METHOD PRIVATE CheckImplementsIList
VAR
	list : List;
    iList : I_List := list;
    result : BOOL;
END_VAR
TEST('ListTests_CheckImplementsIList');

result := iList <> 0;

AssertTrue(Condition := result,
    Message := 'Did not implement IList');

TEST_FINISHED();
END_METHOD

METHOD PUBLIC CheckIsEmptyWhenEmpty
VAR
	result : BOOL;
	list : List;
END_VAR
TEST('CheckIsEmptyWhenEmpty');

// @TEST-RUN
result := list.IsEmpty;

// @TEST-ASSSERT
AssertTrue(
	Condition := result,
	Message := 'Incorrect state of IsEmpty'
);

TEST_FINISHED();
END_METHOD

METHOD PUBLIC CheckIsEmptyWhenFull
VAR
	in : INT := 123;
	result : BOOL;
	list : List;
END_VAR
TEST('CheckIsEmptyWhenFull');

// @TEST-FIXTURE
list.AddItem(in);

// @TEST-RUN
result := list.IsEmpty;

// @TEST-ASSSERT
AssertFalse(
	Condition := result,
	Message := 'Incorrect state of IsEmpty'
);

TEST_FINISHED();
END_METHOD

METHOD PUBLIC CheckOffEvent
VAR
	value : INT := 123;
	list : List;
	handler : CollectionChangedEventHandler(ExpectedOriginator := list);
END_VAR
TEST('CheckOffEvent');

// @TEST-FIXTURE
list.OnEvent('OnChanged',handler);
list.OffEvent('OnChanged',handler);

// @TEST-RUN
list.AddItem(value);

// @TEST-ASSSERT
AssertFalse(
	Condition := handler.EventReceived,
	Message := 'OnceEvent emitted the OnChanged event more than once'
);

TEST_FINISHED();
END_METHOD

METHOD PUBLIC CheckOnceEvent
VAR
	value : INT := 123;
	list : List;
	handler : CollectionChangedEventHandler(ExpectedOriginator := list);
END_VAR
TEST('CheckOnceEvent');

// @TEST-FIXTURE
list.OnceEvent('OnChanged',handler);
list.AddItem(value);
handler.Reset();

// @TEST-RUN
list.AddItem(value);

// @TEST-ASSSERT
AssertFalse(
	Condition := handler.EventReceived,
	Message := 'OnceEvent emitted the OnChanged event more than once'
);

TEST_FINISHED();
END_METHOD

METHOD PUBLIC CheckOnChangedEvent
VAR
	value : INT := 123;
	list : List;
	handler : CollectionChangedEventHandler(ExpectedOriginator := list);
END_VAR
TEST('CheckOnChangedEvent');

// @TEST-FIXTURE
list.OnEvent('OnChanged',handler);

// @TEST-RUN
list.AddItem(value);

// @TEST-ASSSERT
AssertTrue(
	Condition := handler.EventReceived,
	Message := 'Did not emit the OnChanged event'
);

AssertTrue(
	Condition := handler.FromExpectedOriginator,
	Message := 'Did not include itself in the OnChanged event'
);

TEST_FINISHED();
END_METHOD

METHOD PUBLIC CheckOnDisposedEvent
VAR
	pList : POINTER TO List;
	handler : CollectionDisposedEventHandler(ExpectedOriginator := 0);
END_VAR
TEST('CheckOnDisposedEvent');

// @TEST-FIXTURE
pList := __NEW(List);
handler.SetExpectedOriginator(pList^);
pList^.OnEvent('OnDisposed',handler);

// @TEST-RUN
pList^.Dispose();

// @TEST-ASSSERT
AssertTrue(
	Condition := handler.EventReceived,
	Message := 'Did not emit the OnDisposed event'
);

AssertTrue(
	Condition := handler.FromExpectedOriginator,
	Message := 'Did not include itself in the OnDisposed event'
);

TEST_FINISHED();
END_METHOD

METHOD PRIVATE CheckTrimExcessAfterAdding5Items
VAR
	in1 : INT := 1;
	in2 : INT := 2;
	in3 : INT := 3;
	in4 : INT := 4;
	in5 : INT := 5;
	in6 : INT := 6;
	expected : DINT := 5;
	out : DINT;
	list : List;
END_VAR
TEST('CheckTrimExcessAfterAdding5Items');

list.AddItem(in1); // [1, null, null, null]
list.AddItem(in2); // [1, 2, null, null]
list.AddItem(in3); // [1, 2, 3, null]
list.AddItem(in4); // [1, 2, 3, 4]
list.AddItem(in5); // [1, 2, 3, 4, 5, null, null, null]
list.TrimExcess(); // [1, 2, 3, 4, 5]

out := list.Capacity;

AssertEquals(expected, out, 'List was expected to double once 5 items were added');

TEST_FINISHED();
END_METHOD

METHOD PRIVATE CheckTryCopyTo
VAR
	in1 : INT := 123;
	in2 : INT := 456;
	in3 : INT := 789;
	out : ARRAY [0..2] OF INT;
	expected : ARRAY [0..2] OF INT := [123,456,789];
	list : List;
END_VAR
TEST('CheckTryCopyTo');

list.AddItem(in1); // [123]
list.AddItem(in2); // [123,456]
list.AddItem(in3); // [123,456,789]

list.TryCopyTo(out);

AssertEquals(
	Expected := expected,
	Actual := out,
	Message := 'Did not produce the expected result'
);

TEST_FINISHED();
END_METHOD

METHOD PRIVATE CheckTryCopyToLocation
VAR
	in1 : INT := 123;
	in2 : INT := 456;
	in3 : INT := 789;
	out : ARRAY [0..2] OF INT;
	expected : ARRAY [0..2] OF INT := [123,456,789];
	list : List;
END_VAR
TEST('CheckTryCopyToLocation');

list.AddItem(in1); // [123]
list.AddItem(in2); // [123,456]
list.AddItem(in3); // [123,456,789]

list.TryCopyToLocation(ADR(out),SIZEOF(out));

AssertEquals(
	Expected := expected,
	Actual := out,
	Message := 'Did not produce the expected result'
);

TEST_FINISHED();
END_METHOD

METHOD PRIVATE CheckTryInsert
VAR
	in1 : INT := 123;
	in2 : INT := 456;
	in3 : INT := 789;
	out : INT;
	result : BOOL;
	expected : INT := 789;
	list : List;
END_VAR
TEST('CheckTryInsert');

list.AddItem(in1); // [123]
list.AddItem(in1); // [123,456]
list.TryInsert(1, in3); // [123,789,456]

list.TryGetByIndex(1,out);

AssertEquals(expected, out, 'Did not produce the expected result');

TEST_FINISHED();
END_METHOD

METHOD PRIVATE CheckTryRemoveAtInBounds
VAR
	in1 : INT := 123;
	in2 : INT := 456;
	in3 : INT := 789;
	out : INT;
	result : BOOL;
	list : List;
END_VAR
TEST('CheckTryRemoveAtInBounds');

list.AddItem(in1); // [123]
list.AddItem(in2); // [123,456]
list.AddItem(in3); // [123,456,789]

list.TryRemoveAt(0);

result := list.TryGetByIndex(0, out);

AssertTrue(result, 'Couldnt get first item');
AssertEquals(in2, out, 'Array didnt shift up items');

TEST_FINISHED();
END_METHOD

METHOD PRIVATE CheckTryRemoveAtNoItems
VAR
	out : INT;
	result : BOOL;
	list : List;
END_VAR
TEST('CheckTryRemoveAtNoItems');

result := list.TryRemoveAt(0);

AssertFalse(result, 'Returned true while there was nothing to remove');

TEST_FINISHED();
END_METHOD

METHOD PRIVATE CheckTryRemoveAtOutOfBounds
VAR
	in1 : INT := 123;
	in2 : INT := 456;
	in3 : INT := 789;
	out : INT;
	result : BOOL;
	list : List;
END_VAR
TEST('CheckTryRemoveAtOutOfBounds');

list.AddItem(in1); // [123]
list.AddItem(in2); // [123,456]
list.AddItem(in3); // [123,456,789]

result := list.TryRemoveAt(3);

AssertFalse(result, 'Returned true while remove was out of bounds');

TEST_FINISHED();
END_METHOD

METHOD PRIVATE CheckTryRemoveItemFirstShiftUp
VAR
	in1 : INT := 123;
	in2 : INT := 456;
	in3 : INT := 789;
	out : INT;
	result : BOOL;
	expected : INT := 456;
	list : List;
END_VAR
TEST('CheckTryRemoveItemFirstShiftUp');

list.AddItem(in1); // [123]
list.AddItem(in2); // [123,456]
list.AddItem(in3); // [123,456,789]
list.TryRemoveItem(in1); // [456,789]

result := list.TryGetByIndex(0, out);

AssertTrue(result, 'Couldnt get first item');

AssertEquals(expected, out, 'Array didnt shift up items');

TEST_FINISHED();
END_METHOD

METHOD PRIVATE CheckTryRemoveItemNonExisting
VAR
	in1 : INT := 123;
	in2 : INT := 456;
	in3 : INT := 789;
	out : INT;
	result : BOOL;
	list : List;
END_VAR
TEST('CheckTryRemoveItemNonExisting');

list.AddItem(in1); // [123]
list.AddItem(in2); // [123,456]

result := list.TryRemoveItem(in3);

AssertFalse(result, 'RemoveItem returned true which should not happen when item does not exist');

TEST_FINISHED();
END_METHOD

METHOD PRIVATE CheckTryRemoveItemSecondShiftUp
VAR
	in1 : INT := 123;
	in2 : INT := 456;
	in3 : INT := 789;
	out : INT;
	result : BOOL;
	expected : INT := 789;
	list : List;
END_VAR
TEST('CheckTryRemoveItemSecondShiftUp');

list.AddItem(in1); // [123]
list.AddItem(in2); // [123,456]
list.AddItem(in3); // [123,456,789]
list.TryRemoveItem(in2); // [123,789]

result := list.TryGetByIndex(1, out);

AssertTrue(result, 'Coulndt get first item');
AssertEquals(expected, out, 'Array didnt shift up items');

TEST_FINISHED();
END_METHOD

END_FUNCTION_BLOCK

// ---- Tests/ListForwardEnumerator_TestSuite.TcPOU
FUNCTION_BLOCK ListForwardEnumerator_TestSuite EXTENDS TcUnit.FB_TestSuite
VAR
END_VAR

CheckIsValidAtStart();
CheckMoveNextReturnsFalseAtTheEnd();
CheckMoveNextReturnsTrueSingleItem();
CheckMoveNextReturnsFalseWhenEmpty();
CheckMoveNextReturnsTrueMultipleItems();
CheckReset();
CheckTryGet();
CheckTryGetTo();
CheckWorksWithArrays();
CheckWorksWithIntegers();
CheckWorksWithStrings();

METHOD PRIVATE CheckIsValidAtStart
VAR
	result : BOOL;
	store : List;
	enumerator : I_ForwardEnumerator;
END_VAR
TEST('CheckIsValidAtStart');

enumerator := store.GetEnumerator();

result := enumerator.IsValid;
enumerator.Dispose();

AssertTrue(
	Condition := result,
	Message := 'IsValid returned false'
);

TEST_FINISHED();
END_METHOD

METHOD PRIVATE CheckMoveNextReturnsFalseAtTheEnd
VAR
	in1 : INT := 123;
	result : BOOL;
	store : List;
	enumerator : I_ForwardEnumerator;
END_VAR
TEST('CheckMoveNextReturnsFalseAtTheEnd');

store.AddItem(in1);
enumerator := store.GetEnumerator();

enumerator.MoveNext();
result := enumerator.MoveNext();
enumerator.Dispose();

AssertFalse(result,
    'MoveNext did not correctly signal the end of the enumeration');
	
TEST_FINISHED();
END_METHOD

METHOD PRIVATE CheckMoveNextReturnsFalseWhenEmpty
VAR
	result : BOOL;
	store : List;
	enumerator : I_ForwardEnumerator;
	count : DINT;
END_VAR
TEST('CheckMoveNextReturnsFalseWhenEmpty');

count := store.Count;
enumerator := store.GetEnumerator();

result := enumerator.MoveNext();
enumerator.Dispose();

AssertFalse(Condition := result,
    Message := 'MoveNext did not correctly signal the end of the enumeration');

TEST_FINISHED();
END_METHOD

METHOD PRIVATE CheckMoveNextReturnsTrueMultipleItems
VAR
	in1 : INT := 123;
	in2 : INT := 456;
	in3 : INT := 789;
	result : BOOL;
	store : List;
	enumerator : I_ForwardEnumerator;
END_VAR
TEST('CheckMoveNextReturnsTrueMultipleItems');

store.AddItem(in1);
store.AddItem(in2);
store.AddItem(in3);
enumerator := store.GetEnumerator();

result := enumerator.MoveNext();
enumerator.Dispose();

AssertTrue(result, 'MoveNext did not correctly signal there were more items to follow');

TEST_FINISHED();
END_METHOD

METHOD PRIVATE CheckMoveNextReturnsTrueSingleItem
VAR
	in1 : INT := 123;
	result : BOOL;
	store : List;
	enumerator : I_ForwardEnumerator;
END_VAR
TEST('CheckMoveNextReturnsTrueSingleItem');

store.AddItem(in1);
enumerator := store.GetEnumerator();

result := enumerator.MoveNext();
enumerator.Dispose();

AssertTrue(result,
    'MoveNext did not correctly signal there were more items to follow');
	
TEST_FINISHED();
END_METHOD

METHOD PRIVATE CheckReset
VAR
	in1 : ARRAY [0..1] OF REAL := [0.1,2.3];
	in2 : ARRAY [0..1] OF REAL := [1.2,3.4];
	in3 : ARRAY [0..1] OF REAL := [2.3,4.5];
	out : ARRAY [0..1] OF REAL;
	expected : ARRAY [0..1] OF REAL := [0.1,2.3];
	store : List;
	enumerator : I_ForwardEnumerator;
END_VAR
TEST('CheckReset');

store.AddItem(in1);
store.AddItem(in2);
store.AddItem(in3);

enumerator := store.GetEnumerator();

enumerator.MoveNext();
enumerator.MoveNext();
enumerator.Reset();
enumerator.MoveNext();
enumerator.TryGet(out);

enumerator.Dispose();

AssertEquals(
	Expected := expected,
	Actual := out,
	Message := 'Did not produce the expected result'
);

TEST_FINISHED();
END_METHOD

METHOD PRIVATE CheckTryGet
VAR
	in : INT := 123;
	out : INT;
	expected : INT := 123;
	result : BOOL;
	store : List;
	enumerator : I_ForwardEnumerator;
END_VAR
TEST('CheckTryGet');

store.AddItem(in);
enumerator := store.GetEnumerator();
enumerator.MoveNext();

result := enumerator.TryGet(out);
enumerator.Dispose();

AssertTrue(
	Condition := result,
	Message := 'Method returned false'
);

AssertEquals(
	Expected := expected,
	Actual := out,
	Message := 'Did not produce the expected result'
);

TEST_FINISHED();
END_METHOD

METHOD PRIVATE CheckTryGetTo
VAR
	in : INT := 123;
	out : INT;
	expected : INT := 123;
	result : BOOL;
	store : List;
	enumerator : I_ForwardEnumerator;
END_VAR
TEST('CheckTryGetTo');

store.AddItem(in);
enumerator := store.GetEnumerator();
enumerator.MoveNext();

result := enumerator.TryGetTo(ADR(out),SIZEOF(out));
enumerator.Dispose();

AssertTrue(
	Condition := result,
	Message := 'Method returned false'
);

AssertEquals(
	Expected := expected,
	Actual := out,
	Message := 'Did not produce the expected result'
);

TEST_FINISHED();
END_METHOD

METHOD PRIVATE CheckWorksWithArrays
VAR
	in1 : ARRAY [0..1] OF REAL := [0.1,2.3];
	in2 : ARRAY [0..1] OF REAL := [1.2,3.4];
	in3 : ARRAY [0..1] OF REAL := [2.3,4.5];
	out1 : ARRAY [0..1] OF REAL;
	out2 : ARRAY [0..1] OF REAL;
	out3 : ARRAY [0..1] OF REAL;
	expected1 : ARRAY [0..1] OF REAL := [0.1,2.3];
	expected2 : ARRAY [0..1] OF REAL := [1.2,3.4];
	expected3 : ARRAY [0..1] OF REAL := [2.3,4.5];
	store : List;
	enumerator : I_ForwardEnumerator;
END_VAR
TEST('CheckWorksWithArrays');

store.AddItem(in1);
store.AddItem(in2);
store.AddItem(in3);

enumerator := store.GetEnumerator();

enumerator.MoveNext();
enumerator.TryGet(out1);
enumerator.MoveNext();
enumerator.TryGet(out2);
enumerator.MoveNext();
enumerator.TryGet(out3);

enumerator.Dispose();

AssertEquals(
	Expected := expected1,
	Actual := out1,
	Message := 'Did not produce the expected 1st result'
);

AssertEquals(
	Expected := expected2,
	Actual := out2,
	Message := 'Did not produce the expected 2nd result'
);

AssertEquals(
	Expected := expected3,
	Actual := out3,
	Message := 'Did not produce the expected 3rd result'
);

TEST_FINISHED();
END_METHOD

METHOD PRIVATE CheckWorksWithIntegers
VAR
	in1 : INT := 123;
	in2 : INT := 234;
	in3 : INT := 345;
	out1 : INT;
	out2 : INT;
	out3 : INT;
	expected1 : INT := 123;
	expected2 : INT := 234;
	expected3 : INT := 345;
	store : List;
	enumerator : I_ForwardEnumerator;
END_VAR
TEST('CheckWorksWithIntegers');

store.AddItem(in1);
store.AddItem(in2);
store.AddItem(in3);

enumerator := store.GetEnumerator();

enumerator.MoveNext();
enumerator.TryGet(out1);
enumerator.MoveNext();
enumerator.TryGet(out2);
enumerator.MoveNext();
enumerator.TryGet(out3);

enumerator.Dispose();

AssertEquals(
	Expected := expected1,
	Actual := out1,
	Message := 'Did not produce the expected 1st result'
);

AssertEquals(
	Expected := expected2,
	Actual := out2,
	Message := 'Did not produce the expected 2nd result'
);

AssertEquals(
	Expected := expected3,
	Actual := out3,
	Message := 'Did not produce the expected 3rd result'
);

TEST_FINISHED();
END_METHOD

METHOD PRIVATE CheckWorksWithStrings
VAR
	in1 : STRING := 'test1';
	in2 : STRING := 'test2';
	in3 : STRING := 'test3';
	out1 : STRING;
	out2 : STRING;
	out3 : STRING;
	expected1 : STRING := 'test1';
	expected2 : STRING := 'test2';
	expected3 : STRING := 'test3';
	store : List;
	enumerator : I_ForwardEnumerator;
END_VAR
TEST('CheckWorksWithStrings');

store.AddItem(in1);
store.AddItem(in2);
store.AddItem(in3);

enumerator := store.GetEnumerator();

enumerator.MoveNext();
enumerator.TryGet(out1);
enumerator.MoveNext();
enumerator.TryGet(out2);
enumerator.MoveNext();
enumerator.TryGet(out3);

enumerator.Dispose();

AssertEquals(
	Expected := expected1,
	Actual := out1,
	Message := 'Did not produce the expected 1st result'
);

AssertEquals(
	Expected := expected2,
	Actual := out2,
	Message := 'Did not produce the expected 2nd result'
);

AssertEquals(
	Expected := expected3,
	Actual := out3,
	Message := 'Did not produce the expected 3rd result'
);

TEST_FINISHED();
END_METHOD

END_FUNCTION_BLOCK

// ---- Tests/Queue_TestSuite.TcPOU
FUNCTION_BLOCK PUBLIC Queue_TestSuite EXTENDS TcUnit.FB_TestSuite

// check datatypes are handled correctly
CheckListWorksWithIntegers();
CheckListWorksWithStrings();
CheckListWorksWithArrays();

// all other checks
CheckQueueImplementsI_Queue();
CheckContains();
CheckClear();
CheckCount();
CheckAddItem();
CheckTryRemoveItem();
CheckTryDequeueRemovesTheItem();
CheckTryDequeueReturnsTheCorrectValue();
CheckTryPeekReturnsTheCorrectValue();
CheckTryPeekDoesNotRemoveTheItem();
CheckOnChangedEvent();
CheckOnDisposedEvent();
CheckOnceEvent();
CheckOffEvent();
CheckTryCopyTo();
CheckTryCopyToLocation();
CheckQueueOrderIsCorrect();
CheckListReturnsEnumerator();
CheckEnumeratorIsInvalidAfterChange();
CheckIsEmptyWhenEmpty();
CheckIsEmptyWhenFull();

METHOD PUBLIC CheckAddItem
VAR
	in1 : INT := 123;
	in2 : INT := 456;
	in3 : INT := 789;
	result : BOOL;
	queue : Queue;
END_VAR
TEST('CheckAddItem');

// @TEST-FIXTURE
queue.Enqueue(in1); // (lifo->) 123
queue.Enqueue(in2); // (lifo->) 123, 456

// @TEST-RUN
queue.AddItem(in3); // (lifo->) 123, 456, 789
result := queue.Contains(in3);

// @TEST-ASSSERT
AssertTrue(
	Condition := result,
	Message := 'Method returned false'
);

TEST_FINISHED();
END_METHOD

METHOD PUBLIC CheckClear
VAR
	in1 : INT := 123;
	in2 : INT := 456;
	in3 : INT := 789;
	queue : Queue;
END_VAR
TEST('CheckClear');

// @TEST-FIXTURE
queue.Enqueue(in1); // (lifo->) 123
queue.Enqueue(in2); // (lifo->) 123, 456
queue.Enqueue(in2); // (lifo->) 123, 456, 789

// @TEST-RUN
queue.Clear();

// @TEST-ASSSERT
AssertTrue(
	Condition := queue.Count = 0,
	Message := 'The count is not zero'
);

TEST_FINISHED();
END_METHOD

METHOD PUBLIC CheckContains
VAR
	in1 : INT := 123;
	in2 : INT := 456;
	in3 : INT := 789;
	result : BOOL;
	queue : Queue;
END_VAR
TEST('CheckContains');

// @TEST-FIXTURE
queue.Enqueue(in1); // (lifo->) 123
queue.Enqueue(in2); // (lifo->) 123, 456
queue.Enqueue(in2); // (lifo->) 123, 456, 789

// @TEST-RUN
result := queue.Contains(in2);

// @TEST-ASSSERT
AssertTrue(
	Condition := result,
	Message := 'Did not find the item in the queue'
);

TEST_FINISHED();
END_METHOD

METHOD PUBLIC CheckCount
VAR
	in1 : INT := 123;
	in2 : INT := 456;
	in3 : INT := 789;
	total : DINT;
	expected : DINT := 3;
	queue : Queue;
END_VAR
TEST('CheckCount');

// @TEST-FIXTURE
queue.Enqueue(in1); // (lifo->) 123
queue.Enqueue(in2); // (lifo->) 123, 456
queue.Enqueue(in2); // (lifo->) 123, 456, 789

// @TEST-RUN
total := queue.Count;

// @TEST-ASSSERT
AssertEquals(
	Expected := expected,
	Actual := total,
	Message := 'Incorrect count'
);

TEST_FINISHED();
END_METHOD

METHOD PUBLIC CheckEnumeratorIsInvalidAfterChange
VAR
	in : INT := 123;
	result : BOOL;
	queue : Queue;
	enumerator : I_ForwardEnumerator;
END_VAR
TEST('CheckEnumeratorIsInvalidAfterChange');

// @TEST-FIXTURE
enumerator := queue.GetEnumerator();
queue.Enqueue(in);

// @TEST-RUN
result := enumerator.IsValid;
enumerator.Dispose();

// @TEST-ASSSERT
AssertFalse(
	Condition := result,
	Message := 'Method returned true'
);

TEST_FINISHED();
END_METHOD

METHOD PUBLIC CheckIsEmptyWhenEmpty
VAR
	result : BOOL;
	queue : Queue;
END_VAR
TEST('CheckIsEmptyWhenEmpty');

// @TEST-RUN
result := queue.IsEmpty;

// @TEST-ASSSERT
AssertTrue(
	Condition := result,
	Message := 'Incorrect state of IsEmpty'
);

TEST_FINISHED();
END_METHOD

METHOD PUBLIC CheckIsEmptyWhenFull
VAR
	in : INT := 123;
	result : BOOL;
	queue : Queue;
END_VAR
TEST('CheckIsEmptyWhenFull');

// @TEST-FIXTURE
queue.Enqueue(in);

// @TEST-RUN
result := queue.IsEmpty;

// @TEST-ASSSERT
AssertFalse(
	Condition := result,
	Message := 'Incorrect state of IsEmpty'
);

TEST_FINISHED();
END_METHOD

METHOD PUBLIC CheckListReturnsEnumerator
VAR
	in1 : INT := 123;
	in2 : INT := 456;
	in3 : INT := 789;
	enumerator : I_ForwardEnumerator;
	queue : Queue;
END_VAR
TEST('CheckListReturnsEnumerator');

// @TEST-FIXTURE
queue.Enqueue(in1); // (lifo->) 123
queue.Enqueue(in2); // (lifo->) 123, 456
queue.Enqueue(in2); // (lifo->) 123, 456, 789

// @TEST-RUN
enumerator := queue.GetEnumerator();

// @TEST-ASSSERT
AssertTrue(
	Condition := (enumerator <> 0),
	Message := 'Did not return an enumerator'
);

// @TEST-DISPOSE
enumerator.Dispose();

TEST_FINISHED();
END_METHOD

METHOD PUBLIC CheckListWorksWithArrays
VAR
	in : ARRAY [0..1] OF REAL := [0.1,2.3];
	out : ARRAY [0..1] OF REAL;
	expected : ARRAY [0..1] OF REAL := [0.1,2.3];
	result : BOOL;
	queue : Queue;
END_VAR
TEST('CheckListWorksWithArrays');

// @TEST-FIXTURE
queue.Enqueue(in);

// @TEST-RUN
result := queue.TryDequeue(out);

// @TEST-ASSSERT
AssertTrue(
	Condition := result,
	Message := 'Method returned false'
);

AssertEquals(
	Expected := expected,
	Actual := out,
	Message := 'Did not produce the expected result'
);

TEST_FINISHED();
END_METHOD

METHOD PUBLIC CheckListWorksWithIntegers
VAR
	in : INT := 123;
	out : INT;
	expected : INT := 123;
	result : BOOL;
	queue : Queue;
END_VAR
TEST('CheckListWorksWithIntegers');

// @TEST-FIXTURE
queue.Enqueue(in);

// @TEST-RUN
result := queue.TryDequeue(out);

// @TEST-ASSSERT
AssertTrue(
	Condition := result,
	Message := 'Method returned false'
);

AssertEquals(
	Expected := expected,
	Actual := out,
	Message := 'Did not produce the expected result'
);

TEST_FINISHED();
END_METHOD

METHOD PUBLIC CheckListWorksWithStrings
VAR
	in : STRING := 'test';
	out : STRING;
	expected : STRING := 'test';
	result : BOOL;
	queue : Queue;
END_VAR
TEST('CheckListWorksWithStrings');

// @TEST-FIXTURE
queue.Enqueue(in);

// @TEST-RUN
result := queue.TryDequeue(out);

// @TEST-ASSSERT
AssertTrue(
	Condition := result,
	Message := 'Method returned false'
);

AssertEquals(
	Expected := expected,
	Actual := out,
	Message := 'Did not produce the expected result'
);

TEST_FINISHED();
END_METHOD

METHOD PUBLIC CheckOffEvent
VAR
	value : INT := 123;
	queue : queue;
	handler : CollectionChangedEventHandler(ExpectedOriginator := queue);
END_VAR
TEST('CheckOffEvent');

// @TEST-FIXTURE
queue.OnEvent('OnChanged',handler);
queue.OffEvent('OnChanged',handler);

// @TEST-RUN
queue.Enqueue(value);

// @TEST-ASSSERT
AssertFalse(
	Condition := handler.EventReceived,
	Message := 'OnceEvent emitted the OnChanged event more than once'
);

TEST_FINISHED();
END_METHOD

METHOD PUBLIC CheckOnceEvent
VAR
	value : INT := 123;
	queue : Queue;
	handler : CollectionChangedEventHandler(ExpectedOriginator := queue);
END_VAR
TEST('CheckOnceEvent');

// @TEST-FIXTURE
queue.OnceEvent('OnChanged',handler);
queue.Enqueue(value);
handler.Reset();

// @TEST-RUN
queue.Enqueue(value);

// @TEST-ASSSERT
AssertFalse(
	Condition := handler.EventReceived,
	Message := 'OnceEvent emitted the OnChanged event more than once'
);

TEST_FINISHED();
END_METHOD

METHOD PUBLIC CheckOnChangedEvent
VAR
	value : INT := 123;
	queue : Queue;
	handler : CollectionChangedEventHandler(ExpectedOriginator := queue);
END_VAR
TEST('CheckOnChangedEvent');

// @TEST-FIXTURE
queue.OnEvent('OnChanged', handler);

// @TEST-RUN
queue.Enqueue(value);

// @TEST-ASSSERT
AssertTrue(
	Condition := handler.EventReceived,
	Message := 'Did not emit the OnChanged event'
);

AssertTrue(
	Condition := handler.FromExpectedOriginator,
	Message := 'Did not include itself in the OnChanged event'
);

TEST_FINISHED();
END_METHOD

METHOD PUBLIC CheckOnDisposedEvent
VAR
	value : INT := 123;
	pQueue : POINTER TO Queue;
	handler : CollectionDisposedEventHandler(ExpectedOriginator := 0);
END_VAR
TEST('CheckOnDisposedEvent');

// @TEST-FIXTURE
pQueue := __NEW(Queue);
handler.SetExpectedOriginator(pQueue^);
pQueue^.OnEvent('OnDisposed', handler);

// @TEST-RUN
pQueue^.Dispose();

// @TEST-ASSSERT
AssertTrue(
	Condition := handler.EventReceived,
	Message := 'Did not emit the OnDisposed event'
);

AssertTrue(
	Condition := handler.FromExpectedOriginator,
	Message := 'Did not include itself in the OnDisposed event'
);

TEST_FINISHED();
END_METHOD

METHOD PUBLIC CheckQueueImplementsI_Queue
VAR
	queue : Queue;
    iQueue : I_Queue := queue;
    result : BOOL;
END_VAR
TEST('CheckQueueImplementsI_Queue');

// @TEST-FIXTURE

// @TEST-RUN
result := iQueue <> 0;

// @TEST-ASSSERT
AssertTrue(
	Condition := result,
	Message := 'Did not implement I_Queue'
);

TEST_FINISHED();
END_METHOD

METHOD PUBLIC CheckQueueOrderIsCorrect
VAR
	in1 : INT := 123;
	in2 : INT := 456;
	in3 : INT := 789;
	out1, out2, out3 : INT;
	expected1 : INT := 123;
	expected2 : INT := 456;
	expected3 : INT := 789;
	result1, result2, result3 : BOOL;
	queue : Queue;
END_VAR
TEST('CheckQueueOrderIsCorrect');

// @TEST-FIXTURE
queue.Enqueue(in1); // (lifo->) 123
queue.Enqueue(in2); // (lifo->) 123, 456
queue.Enqueue(in3); // (lifo->) 123, 456, 789

// @TEST-RUN
result1 := queue.TryDequeue(out1); // (lifo->) 456, 789
result2 := queue.TryDequeue(out2); // (lifo->) 789
result3 := queue.TryDequeue(out3); // (lifo->) 

// @TEST-ASSSERT
AssertTrue(
	Condition := result1 AND result2 AND result3,
	Message := 'Method returned false'
);

AssertEquals(
	Expected := expected1,
	Actual := out1,
	Message := 'Did not produce the expected result'
);

AssertEquals(
	Expected := expected2,
	Actual := out2,
	Message := 'Did not produce the expected result'
);

AssertEquals(
	Expected := expected3,
	Actual := out3,
	Message := 'Did not produce the expected result'
);

TEST_FINISHED();
END_METHOD

METHOD PUBLIC CheckTryCopyTo
VAR
	in1 : INT := 123;
	in2 : INT := 456;
	in3 : INT := 789;
	out : ARRAY [0..2] OF INT;
	expected : ARRAY [0..2] OF INT := [123,456,789];
	queue : Queue;
END_VAR
TEST('CheckTryCopyTo');

// @TEST-FIXTURE
queue.Enqueue(in1); // (lifo->) 123
queue.Enqueue(in2); // (lifo->) 123, 456
queue.Enqueue(in3); // (lifo->) 123, 456, 789

// @TEST-RUN
queue.TryCopyTo(out);

// @TEST-ASSSERT
AssertEquals(
	Expected := expected,
	Actual := out,
	Message := 'Did not produce the expected result'
);

TEST_FINISHED();
END_METHOD

METHOD PUBLIC CheckTryCopyToLocation
VAR
	in1 : INT := 123;
	in2 : INT := 456;
	in3 : INT := 789;
	out : ARRAY [0..2] OF INT;
	expected : ARRAY [0..2] OF INT := [123,456,789];
	queue : Queue;
END_VAR
TEST('CheckTryCopyToLocation');

// @TEST-FIXTURE
queue.Enqueue(in1); // (lifo->) 123
queue.Enqueue(in2); // (lifo->) 123, 456
queue.Enqueue(in3); // (lifo->) 123, 456, 789

// @TEST-RUN
queue.TryCopyToLocation(ADR(out),SIZEOF(out));

// @TEST-ASSSERT
AssertEquals(
	Expected := expected,
	Actual := out,
	Message := 'Did not produce the expected result'
);

TEST_FINISHED();
END_METHOD

METHOD PUBLIC CheckTryDequeueRemovesTheItem
VAR
	in : INT := 123;
	out : INT;
	total : DINT;
	expected : DINT := 0;
	queue : Queue;
END_VAR
TEST('CheckTryDequeueDoesNotRemoveTheItem');

// @TEST-FIXTURE
queue.Enqueue(in); // (lifo->) 123

// @TEST-RUN
queue.TryDequeue(out);
total := queue.Count;

// @TEST-ASSSERT
AssertEquals(
	Expected := expected,
	Actual := total,
	Message := 'Incorrect count'
);

TEST_FINISHED();
END_METHOD

METHOD PUBLIC CheckTryDequeueReturnsTheCorrectValue
VAR
	in : INT := 123;
	out : INT;
	expected : INT := 123;
	result : BOOL;
	queue : Queue;
END_VAR
TEST('CheckTryDequeueReturnsTheCorrectValue');

// @TEST-FIXTURE
queue.Enqueue(in);

// @TEST-RUN
result := queue.TryPeek(out);

// @TEST-ASSSERT
AssertTrue(
	Condition := result,
	Message := 'Method returned false'
);

AssertEquals(
	Expected := expected,
	Actual := out,
	Message := 'Did not produce the expected result'
);

TEST_FINISHED();
END_METHOD

METHOD PUBLIC CheckTryPeekDoesNotRemoveTheItem
VAR
	in : INT := 123;
	out : INT;
	total : DINT;
	expected : DINT := 1;
	queue : Queue;
END_VAR
TEST('CheckTryPeekDoesNotRemoveTheItem');

// @TEST-FIXTURE
queue.Enqueue(in); // (lifo->) 123

// @TEST-RUN
queue.TryPeek(out);
total := queue.Count;

// @TEST-ASSSERT
AssertEquals(
	Expected := expected,
	Actual := total,
	Message := 'Incorrect count'
);

TEST_FINISHED();
END_METHOD

METHOD PUBLIC CheckTryPeekReturnsTheCorrectValue
VAR
	in : INT := 123;
	out : INT;
	expected : INT := 123;
	result : BOOL;
	queue : Queue;
END_VAR
TEST('CheckTryPeekReturnsTheCorrectValue');

// @TEST-FIXTURE
queue.Enqueue(in);

// @TEST-RUN
result := queue.TryPeek(out);

// @TEST-ASSSERT
AssertTrue(
	Condition := result,
	Message := 'Method returned false'
);

AssertEquals(
	Expected := expected,
	Actual := out,
	Message := 'Did not produce the expected result'
);

TEST_FINISHED();
END_METHOD

METHOD PUBLIC CheckTryRemoveItem
VAR
	in1 : INT := 123;
	in2 : INT := 456;
	in3 : INT := 789;
	result : BOOL;
	queue : Queue;
END_VAR
TEST('CheckTryRemoveItem');

// @TEST-FIXTURE
queue.Enqueue(in1); // (lifo->) 123
queue.Enqueue(in2); // (lifo->) 123, 456
queue.Enqueue(in3); // (lifo->) 123, 456, 789

// @TEST-RUN
queue.TryRemoveItem(in2); // (lifo->) 123, 789
result := queue.Contains(in2);

// @TEST-ASSSERT
AssertFalse(
	Condition := result,
	Message := 'Method returned true'
);

TEST_FINISHED();
END_METHOD

END_FUNCTION_BLOCK

// ---- Tests/QueueForwardEnumerator_TestSuite.TcPOU
FUNCTION_BLOCK PUBLIC QueueForwardEnumerator_TestSuite EXTENDS TcUnit.FB_TestSuite

CheckIsValidAtStart();
CheckMoveNextReturnsFalseAtTheEnd();
CheckMoveNextReturnsFalseWhenEmpty();
CheckMoveNextReturnsTrueMultipleItems();
CheckMoveNextReturnsTrueSingleItem();
CheckReset();
CheckTryGet();
CheckTryGetTo();
CheckWorksWithIntegers();
CheckWorksWithStrings();
CheckWorksWithArrays();

METHOD PUBLIC CheckIsValidAtStart
VAR
	result : BOOL;
	queue : Queue;
	enumerator : I_ForwardEnumerator;
END_VAR
TEST('CheckIsValidAtStart');

enumerator := queue.GetEnumerator();

result := enumerator.IsValid;
enumerator.Dispose();

AssertTrue(
	Condition := result,
	Message := 'Method returned false'
);

TEST_FINISHED();
END_METHOD

METHOD PRIVATE CheckMoveNextReturnsFalseAtTheEnd
VAR
	in1 : INT := 123;
	result : BOOL;
	queue : Queue;
	enumerator : I_ForwardEnumerator;
END_VAR
TEST('CheckMoveNextReturnsFalseAtTheEnd');

queue.Enqueue(in1);
enumerator := queue.GetEnumerator();

enumerator.MoveNext();
result := enumerator.MoveNext();
enumerator.Dispose();

AssertFalse(result,
    'MoveNext did not correctly signal the end of the enumeration');
	
TEST_FINISHED();
END_METHOD

METHOD PUBLIC CheckMoveNextReturnsFalseWhenEmpty
VAR
	result : BOOL;
	queue : Queue;
	enumerator : I_ForwardEnumerator;
END_VAR
TEST('CheckMoveNextReturnsFalseWhenEmpty');

enumerator := queue.GetEnumerator();

result := enumerator.MoveNext();
enumerator.Dispose();

AssertFalse(
	Condition := result,
	Message := 'MoveNext did not correctly signal the end of the enumeration'
);

TEST_FINISHED();
END_METHOD

METHOD PRIVATE CheckMoveNextReturnsTrueMultipleItems
VAR
	in1 : INT := 123;
	in2 : INT := 456;
	in3 : INT := 789;
	result : BOOL;
	queue : Queue;
	enumerator : I_ForwardEnumerator;
END_VAR
TEST('CheckMoveNextReturnsTrueMultipleItems');

queue.Enqueue(in1);
queue.Enqueue(in2);
queue.Enqueue(in3);
enumerator := queue.GetEnumerator();

result := enumerator.MoveNext();
enumerator.Dispose();

AssertTrue(result, 'MoveNext did not correctly signal there were more items to follow');

TEST_FINISHED();
END_METHOD

METHOD PRIVATE CheckMoveNextReturnsTrueSingleItem
VAR
	in1 : INT := 123;
	result : BOOL;
	queue : Queue;
	enumerator : I_ForwardEnumerator;
END_VAR
TEST('CheckMoveNextReturnsTrueSingleItem');

queue.Enqueue(in1);
enumerator := queue.GetEnumerator();

result := enumerator.MoveNext();
enumerator.Dispose();

AssertTrue(result,
    'MoveNext did not correctly signal there were more items to follow');
	
TEST_FINISHED();
END_METHOD

METHOD PUBLIC CheckReset
VAR
	in1 : ARRAY [0..1] OF REAL := [0.1,2.3];
	in2 : ARRAY [0..1] OF REAL := [1.2,3.4];
	in3 : ARRAY [0..1] OF REAL := [2.3,4.5];
	out : ARRAY [0..1] OF REAL;
	expected : ARRAY [0..1] OF REAL := [0.1,2.3];
	queue : Queue;
	enumerator : I_ForwardEnumerator;
END_VAR
TEST('CheckReset');

queue.Enqueue(in1);
queue.Enqueue(in2);
queue.Enqueue(in3);

enumerator := queue.GetEnumerator();

enumerator.MoveNext();
enumerator.MoveNext();
enumerator.Reset();
enumerator.MoveNext();
enumerator.TryGet(out);

enumerator.Dispose();

AssertEquals(
	Expected := expected,
	Actual := out,
	Message := 'Did not produce the expected result'
);

TEST_FINISHED();
END_METHOD

METHOD PUBLIC CheckTryGet
VAR
	in : INT := 123;
	out : INT;
	expected : INT := 123;
	result : BOOL;
	queue : Queue;
	enumerator : I_ForwardEnumerator;
END_VAR
TEST('CheckTryGet');

queue.Enqueue(in);
enumerator := queue.GetEnumerator();
enumerator.MoveNext();

result := enumerator.TryGet(out);
enumerator.Dispose();

AssertTrue(
	Condition := result,
	Message := 'Method returned false'
);

AssertEquals(
	Expected := expected,
	Actual := out,
	Message := 'Did not produce the expected result'
);

TEST_FINISHED();
END_METHOD

METHOD PUBLIC CheckTryGetTo
VAR
	in : INT := 123;
	out : INT;
	expected : INT := 123;
	result : BOOL;
	queue : Queue;
	enumerator : I_ForwardEnumerator;
END_VAR
TEST('CheckTryGetTo');

queue.Enqueue(in);
enumerator := queue.GetEnumerator();
enumerator.MoveNext();

result := enumerator.TryGetTo(ADR(out),SIZEOF(out));
enumerator.Dispose();

AssertTrue(
	Condition := result,
	Message := 'Method returned false'
);

AssertEquals(
	Expected := expected,
	Actual := out,
	Message := 'Did not produce the expected result'
);

TEST_FINISHED();
END_METHOD

METHOD PUBLIC CheckWorksWithArrays
VAR
	in1 : ARRAY [0..1] OF REAL := [0.1,2.3];
	in2 : ARRAY [0..1] OF REAL := [1.2,3.4];
	in3 : ARRAY [0..1] OF REAL := [2.3,4.5];
	out1 : ARRAY [0..1] OF REAL;
	out2 : ARRAY [0..1] OF REAL;
	out3 : ARRAY [0..1] OF REAL;
	expected1 : ARRAY [0..1] OF REAL := [0.1,2.3];
	expected2 : ARRAY [0..1] OF REAL := [1.2,3.4];
	expected3 : ARRAY [0..1] OF REAL := [2.3,4.5];
	queue : Queue;
	enumerator : I_ForwardEnumerator;
END_VAR
TEST('CheckWorksWithArrays');

queue.Enqueue(in1);
queue.Enqueue(in2);
queue.Enqueue(in3);

enumerator := queue.GetEnumerator();

enumerator.MoveNext();
enumerator.TryGet(out1);
enumerator.MoveNext();
enumerator.TryGet(out2);
enumerator.MoveNext();
enumerator.TryGet(out3);

enumerator.Dispose();

AssertEquals(
	Expected := expected1,
	Actual := out1,
	Message := 'Did not produce the expected 1st result'
);

AssertEquals(
	Expected := expected2,
	Actual := out2,
	Message := 'Did not produce the expected 2nd result'
);

AssertEquals(
	Expected := expected3,
	Actual := out3,
	Message := 'Did not produce the expected 3rd result'
);

TEST_FINISHED();
END_METHOD

METHOD PUBLIC CheckWorksWithIntegers
VAR
	in1 : INT := 123;
	in2 : INT := 234;
	in3 : INT := 345;
	out1 : INT;
	out2 : INT;
	out3 : INT;
	expected1 : INT := 123;
	expected2 : INT := 234;
	expected3 : INT := 345;
	queue : Queue;
	enumerator : I_ForwardEnumerator;
END_VAR
TEST('CheckWorksWithIntegers');

queue.Enqueue(in1);
queue.Enqueue(in2);
queue.Enqueue(in3);

enumerator := queue.GetEnumerator();

enumerator.MoveNext();
enumerator.TryGet(out1);
enumerator.MoveNext();
enumerator.TryGet(out2);
enumerator.MoveNext();
enumerator.TryGet(out3);

enumerator.Dispose();

AssertEquals(
	Expected := expected1,
	Actual := out1,
	Message := 'Did not produce the expected 1st result'
);

AssertEquals(
	Expected := expected2,
	Actual := out2,
	Message := 'Did not produce the expected 2nd result'
);

AssertEquals(
	Expected := expected3,
	Actual := out3,
	Message := 'Did not produce the expected 3rd result'
);

TEST_FINISHED();
END_METHOD

METHOD PUBLIC CheckWorksWithStrings
VAR
	in1 : STRING := 'test1';
	in2 : STRING := 'test2';
	in3 : STRING := 'test3';
	out1 : STRING;
	out2 : STRING;
	out3 : STRING;
	expected1 : STRING := 'test1';
	expected2 : STRING := 'test2';
	expected3 : STRING := 'test3';
	queue : Queue;
	enumerator : I_ForwardEnumerator;
END_VAR
TEST('CheckWorksWithStrings');

queue.Enqueue(in1);
queue.Enqueue(in2);
queue.Enqueue(in3);

enumerator := queue.GetEnumerator();

enumerator.MoveNext();
enumerator.TryGet(out1);
enumerator.MoveNext();
enumerator.TryGet(out2);
enumerator.MoveNext();
enumerator.TryGet(out3);

enumerator.Dispose();

AssertEquals(
	Expected := expected1,
	Actual := out1,
	Message := 'Did not produce the expected 1st result'
);

AssertEquals(
	Expected := expected2,
	Actual := out2,
	Message := 'Did not produce the expected 2nd result'
);

AssertEquals(
	Expected := expected3,
	Actual := out3,
	Message := 'Did not produce the expected 3rd result'
);

TEST_FINISHED();
END_METHOD

END_FUNCTION_BLOCK

// ---- Tests/Stack_TestSuite.TcPOU
FUNCTION_BLOCK PUBLIC Stack_TestSuite EXTENDS TcUnit.FB_TestSuite

// check datatypes are handled correctly
CheckListWorksWithIntegers();
CheckListWorksWithStrings();
CheckListWorksWithArrays();

// all other checks
CheckStackImplementsI_Stack();
CheckContains();
CheckClear();
CheckCount();
CheckAddItem();
CheckTryRemoveItem();
CheckTryPopRemovesTheItem();
CheckTryPopReturnsTheCorrectValue();
CheckTryPeekReturnsTheCorrectValue();
CheckTryPeekDoesNotRemoveTheItem();
CheckOnChangedEvent();
CheckOnDisposedEvent();
CheckOnceEvent();
CheckOffEvent();
CheckTryCopyTo();
CheckTryCopyToLocation();
CheckStackOrderIsCorrect();
CheckListReturnsEnumerator();
CheckEnumeratorIsInvalidAfterChange();
CheckIsEmptyWhenEmpty();
CheckIsEmptyWhenFull();

METHOD PUBLIC CheckAddItem
VAR
	in1 : INT := 123;
	in2 : INT := 456;
	in3 : INT := 789;
	result : BOOL;
	stack : Stack;
END_VAR
TEST('CheckAddItem');

// @TEST-FIXTURE
stack.Push(in1); // (fifo->) 123
stack.Push(in2); // (fifo->) 456, 123

// @TEST-RUN
stack.AddItem(in3); // fifo->) 789, 456, 123
result := stack.Contains(in3);

// @TEST-ASSSERT
AssertTrue(
	Condition := result,
	Message := 'Method returned false'
);

TEST_FINISHED();
END_METHOD

METHOD PUBLIC CheckClear
VAR
	in1 : INT := 123;
	in2 : INT := 456;
	in3 : INT := 789;
	stack : Stack;
END_VAR
TEST('CheckClear');

// @TEST-FIXTURE
stack.Push(in1); // (fifo->) 123
stack.Push(in2); // (fifo->) 456, 123
stack.Push(in2); // (fifo->) 789, 456, 123

// @TEST-RUN
stack.Clear();

// @TEST-ASSSERT
AssertTrue(
	Condition := stack.Count = 0,
	Message := 'The count is not zero'
);

TEST_FINISHED();
END_METHOD

METHOD PUBLIC CheckContains
VAR
	in1 : INT := 123;
	in2 : INT := 456;
	in3 : INT := 789;
	result : BOOL;
	stack : Stack;
END_VAR
TEST('CheckContains');

// @TEST-FIXTURE
stack.Push(in1); // (fifo->) 123
stack.Push(in2); // (fifo->) 456, 123
stack.Push(in2); // (fifo->) 789, 456, 123

// @TEST-RUN
result := stack.Contains(in2);

// @TEST-ASSSERT
AssertTrue(
	Condition := result,
	Message := 'Did not find the item in the queue'
);

TEST_FINISHED();
END_METHOD

METHOD PUBLIC CheckCount
VAR
	in1 : INT := 123;
	in2 : INT := 456;
	in3 : INT := 789;
	total : DINT;
	expected : DINT := 3;
	stack : Stack;
END_VAR
TEST('CheckCount');

// @TEST-FIXTURE
stack.Push(in1); // (fifo->) 123
stack.Push(in2); // (fifo->) 456, 123
stack.Push(in2); // (fifo->) 789, 456, 123

// @TEST-RUN
total := stack.Count;

// @TEST-ASSSERT
AssertEquals(
	Expected := expected,
	Actual := total,
	Message := 'Incorrect count'
);

TEST_FINISHED();
END_METHOD

METHOD PUBLIC CheckEnumeratorIsInvalidAfterChange
VAR
	in : INT := 123;
	result : BOOL;
	stack : Stack;
	enumerator : I_ForwardEnumerator;
END_VAR
TEST('CheckEnumeratorIsInvalidAfterChange');

// @TEST-FIXTURE
enumerator := stack.GetEnumerator();
stack.Push(in);

// @TEST-RUN
result := enumerator.IsValid;
enumerator.Dispose();

// @TEST-ASSSERT
AssertFalse(
	Condition := result,
	Message := 'Method returned true'
);

TEST_FINISHED();
END_METHOD

METHOD PUBLIC CheckIsEmptyWhenEmpty
VAR
	result : BOOL;
	stack : Stack;
END_VAR
TEST('CheckIsEmptyWhenEmpty');

// @TEST-RUN
result := stack.IsEmpty;

// @TEST-ASSSERT
AssertTrue(
	Condition := result,
	Message := 'Incorrect state of IsEmpty'
);

TEST_FINISHED();
END_METHOD

METHOD PUBLIC CheckIsEmptyWhenFull
VAR
	in : INT := 123;
	result : BOOL;
	stack : Stack;
END_VAR
TEST('CheckIsEmptyWhenFull');

// @TEST-FIXTURE
stack.Push(in);

// @TEST-RUN
result := stack.IsEmpty;

// @TEST-ASSSERT
AssertFalse(
	Condition := result,
	Message := 'Incorrect state of IsEmpty'
);

TEST_FINISHED();
END_METHOD

METHOD PUBLIC CheckListReturnsEnumerator
VAR
	in1 : INT := 123;
	in2 : INT := 456;
	in3 : INT := 789;
	enumerator : I_ForwardEnumerator;
	stack : Stack;
END_VAR
TEST('CheckListReturnsEnumerator');

// @TEST-FIXTURE
stack.Push(in1); // (fifo->) 123
stack.Push(in2); // (fifo->) 456, 123
stack.Push(in2); // (fifo->) 789, 456, 123

// @TEST-RUN
enumerator := stack.GetEnumerator();

// @TEST-ASSSERT
AssertTrue(
	Condition := (enumerator <> 0),
	Message := 'Did not return an enumerator'
);

// @TEST-DISPOSE
enumerator.Dispose();

TEST_FINISHED();
END_METHOD

METHOD PUBLIC CheckListWorksWithArrays
VAR
	in : ARRAY [0..1] OF REAL := [0.1,2.3];
	out : ARRAY [0..1] OF REAL;
	expected : ARRAY [0..1] OF REAL := [0.1,2.3];
	result : BOOL;
	stack : Stack;
END_VAR
TEST('CheckListWorksWithArrays');

// @TEST-FIXTURE
stack.Push(in);

// @TEST-RUN
result := stack.TryPop(out);

// @TEST-ASSSERT
AssertTrue(
	Condition := result,
	Message := 'Method returned false'
);

AssertEquals(
	Expected := expected,
	Actual := out,
	Message := 'Did not produce the expected result'
);

TEST_FINISHED();
END_METHOD

METHOD PUBLIC CheckListWorksWithIntegers
VAR
	in : INT := 123;
	out : INT;
	expected : INT := 123;
	result : BOOL;
	stack : Stack;
END_VAR
TEST('CheckListWorksWithIntegers');

// @TEST-FIXTURE
stack.Push(in);

// @TEST-RUN
result := stack.TryPop(out);

// @TEST-ASSSERT
AssertTrue(
	Condition := result,
	Message := 'Method returned false'
);

AssertEquals(
	Expected := expected,
	Actual := out,
	Message := 'Did not produce the expected result'
);

TEST_FINISHED();
END_METHOD

METHOD PUBLIC CheckListWorksWithStrings
VAR
	in : STRING := 'test';
	out : STRING;
	expected : STRING := 'test';
	result : BOOL;
	stack : Stack;
END_VAR
TEST('CheckListWorksWithStrings');

// @TEST-FIXTURE
stack.Push(in);

// @TEST-RUN
result := stack.TryPop(out);

// @TEST-ASSSERT
AssertTrue(
	Condition := result,
	Message := 'Method returned false'
);

AssertEquals(
	Expected := expected,
	Actual := out,
	Message := 'Did not produce the expected result'
);

TEST_FINISHED();
END_METHOD

METHOD PUBLIC CheckOffEvent
VAR
	value : INT := 123;
	stack : Stack;
	handler : CollectionChangedEventHandler(ExpectedOriginator := stack);
END_VAR
TEST('CheckOffEvent');

// @TEST-FIXTURE
stack.OnEvent('OnChanged',handler);
stack.OffEvent('OnChanged',handler);

// @TEST-RUN
stack.Push(value);

// @TEST-ASSSERT
AssertFalse(
	Condition := handler.EventReceived,
	Message := 'OnceEvent emitted the OnChanged event more than once'
);

TEST_FINISHED();
END_METHOD

METHOD PUBLIC CheckOnceEvent
VAR
	value : INT := 123;
	stack : Stack;
	handler : CollectionChangedEventHandler(ExpectedOriginator := stack);
END_VAR
TEST('CheckOnceEvent');

// @TEST-FIXTURE
stack.OnceEvent('OnChanged',handler);
stack.Push(value);
handler.Reset();

// @TEST-RUN
stack.Push(value);

// @TEST-ASSSERT
AssertFalse(
	Condition := handler.EventReceived,
	Message := 'OnceEvent emitted the OnChanged event more than once'
);

TEST_FINISHED();
END_METHOD

METHOD PUBLIC CheckOnChangedEvent
VAR
	value : INT := 123;
	stack : Stack;
	handler : CollectionChangedEventHandler(ExpectedOriginator := stack);
END_VAR
TEST('CheckOnChangedEvent');

// @TEST-FIXTURE
stack.OnEvent('OnChanged',handler);

// @TEST-RUN
stack.Push(value);

// @TEST-ASSSERT
AssertTrue(
	Condition := handler.EventReceived,
	Message := 'Did not emit the OnChanged event'
);

AssertTrue(
	Condition := handler.FromExpectedOriginator,
	Message := 'Did not include itself in the OnChanged event'
);

TEST_FINISHED();
END_METHOD

METHOD PUBLIC CheckOnDisposedEvent
VAR
	value : INT := 123;
	pStack : POINTER TO Stack;
	handler : CollectionDisposedEventHandler(ExpectedOriginator := 0);
END_VAR
TEST('CheckOnDisposedEvent');

// @TEST-FIXTURE
pStack := __NEW(Stack);
handler.SetExpectedOriginator(pStack^);
pStack^.OnEvent('OnDisposed',handler);

// @TEST-RUN
pStack^.Dispose();

// @TEST-ASSSERT
AssertTrue(
	Condition := handler.EventReceived,
	Message := 'Did not emit the OnDisposed event'
);

AssertTrue(
	Condition := handler.FromExpectedOriginator,
	Message := 'Did not include itself in the OnDisposed event'
);

TEST_FINISHED();
END_METHOD

METHOD PUBLIC CheckStackImplementsI_Stack
VAR
	stack : Stack;
    iStack : I_Stack := stack;
    result : BOOL;
END_VAR
TEST('CheckStackImplementsI_Stack');

// @TEST-FIXTURE

// @TEST-RUN
result := iStack <> 0;

// @TEST-ASSSERT
AssertTrue(
	Condition := result,
	Message := 'Did not implement I_Stack'
);

TEST_FINISHED();
END_METHOD

METHOD PUBLIC CheckStackOrderIsCorrect
VAR
	in1 : INT := 123;
	in2 : INT := 456;
	in3 : INT := 789;
	out1, out2, out3 : INT;
	expected1 : INT := 789;
	expected2 : INT := 456;
	expected3 : INT := 123;
	result1, result2, result3 : BOOL;
	stack : Stack;
END_VAR
TEST('CheckStackOrderIsCorrect');

// @TEST-FIXTURE
stack.Push(in1); // (fifo->) 123
stack.Push(in2); // (fifo->) 456, 123
stack.Push(in3); // (fifo->) 789, 456, 123

// @TEST-RUN
result1 := stack.TryPop(out1);
result2 := stack.TryPop(out2);
result3 := stack.TryPop(out3);

// @TEST-ASSSERT
AssertTrue(
	Condition := result1 AND result2 AND result3,
	Message := 'Method returned false'
);

AssertEquals(
	Expected := expected1,
	Actual := out1,
	Message := 'Did not produce the expected result'
);

AssertEquals(
	Expected := expected2,
	Actual := out2,
	Message := 'Did not produce the expected result'
);

AssertEquals(
	Expected := expected3,
	Actual := out3,
	Message := 'Did not produce the expected result'
);

TEST_FINISHED();
END_METHOD

METHOD PUBLIC CheckTryCopyTo
VAR
	in1 : INT := 123;
	in2 : INT := 456;
	in3 : INT := 789;
	out : ARRAY [0..2] OF INT;
	expected : ARRAY [0..2] OF INT := [789,456,123];
	stack : Stack;
END_VAR
TEST('CheckTryCopyTo');

// @TEST-FIXTURE
stack.Push(in1); // (fifo->) 123
stack.Push(in2); // (fifo->) 456, 123
stack.Push(in3); // (fifo->) 789, 456, 123

// @TEST-RUN
stack.TryCopyTo(out);

// @TEST-ASSSERT
AssertEquals(
	Expected := expected,
	Actual := out,
	Message := 'Did not produce the expected result'
);

TEST_FINISHED();
END_METHOD

METHOD PUBLIC CheckTryCopyToLocation
VAR
	in1 : INT := 123;
	in2 : INT := 456;
	in3 : INT := 789;
	out : ARRAY [0..2] OF INT;
	expected : ARRAY [0..2] OF INT := [789,456,123];
	stack : Stack;
END_VAR
TEST('CheckTryCopyToLocation');

// @TEST-FIXTURE
stack.Push(in1); // (fifo->) 123
stack.Push(in2); // (fifo->) 456, 123
stack.Push(in3); // (fifo->) 789, 456, 123

// @TEST-RUN
stack.TryCopyToLocation(ADR(out),SIZEOF(out));

// @TEST-ASSSERT
AssertEquals(
	Expected := expected,
	Actual := out,
	Message := 'Did not produce the expected result'
);

TEST_FINISHED();
END_METHOD

METHOD PUBLIC CheckTryPeekDoesNotRemoveTheItem
VAR
	in : INT := 123;
	out : INT;
	total : DINT;
	expected : DINT := 1;
	stack : Stack;
END_VAR
TEST('CheckTryPeekDoesNotRemoveTheItem');

// @TEST-FIXTURE
stack.Push(in); // (fifo->) 123

// @TEST-RUN
stack.TryPeek(out);
total := stack.Count;

// @TEST-ASSSERT
AssertEquals(
	Expected := expected,
	Actual := total,
	Message := 'Incorrect count'
);

TEST_FINISHED();
END_METHOD

METHOD PUBLIC CheckTryPeekReturnsTheCorrectValue
VAR
	in : INT := 123;
	out : INT;
	expected : INT := 123;
	result : BOOL;
	stack : Stack;
END_VAR
TEST('CheckTryPeekReturnsTheCorrectValue');

// @TEST-FIXTURE
stack.Push(in); // (fifo->) 123

// @TEST-RUN
result := stack.TryPeek(out);

// @TEST-ASSSERT
AssertTrue(
	Condition := result,
	Message := 'Method returned false'
);

AssertEquals(
	Expected := expected,
	Actual := out,
	Message := 'Did not produce the expected result'
);

TEST_FINISHED();
END_METHOD

METHOD PUBLIC CheckTryPopRemovesTheItem
VAR
	in : INT := 123;
	out : INT;
	total : DINT;
	expected : DINT := 0;
	stack : Stack;
END_VAR
TEST('CheckTryPopRemovesTheItem');

// @TEST-FIXTURE
stack.Push(in); // (fifo->) 123

// @TEST-RUN
stack.TryPop(out);
total := stack.Count;

// @TEST-ASSSERT
AssertEquals(
	Expected := expected,
	Actual := total,
	Message := 'Incorrect count'
);

TEST_FINISHED();
END_METHOD

METHOD PUBLIC CheckTryPopReturnsTheCorrectValue
VAR
	in : INT := 123;
	out : INT;
	expected : INT := 123;
	result : BOOL;
	stack : Stack;
END_VAR
TEST('CheckTryDequeueReturnsTheCorrectValue');

// @TEST-FIXTURE
stack.Push(in); // (fifo->) 123

// @TEST-RUN
result := stack.TryPop(out);

// @TEST-ASSSERT
AssertTrue(
	Condition := result,
	Message := 'Method returned false'
);

AssertEquals(
	Expected := expected,
	Actual := out,
	Message := 'Did not produce the expected result'
);

TEST_FINISHED();
END_METHOD

METHOD PUBLIC CheckTryRemoveItem
VAR
	in1 : INT := 123;
	in2 : INT := 456;
	in3 : INT := 789;
	result : BOOL;
	stack : Stack;
END_VAR
TEST('CheckTryRemoveItem');

// @TEST-FIXTURE
stack.Push(in1); // (fifo->) 123
stack.Push(in2); // (fifo->) 456, 123
stack.Push(in3); // (fifo->) 789, 456, 123

// @TEST-RUN
stack.TryRemoveItem(in2); // (lifo->) 789, 123
result := stack.Contains(in2);

// @TEST-ASSSERT
AssertFalse(
	Condition := result,
	Message := 'Method returned true'
);

TEST_FINISHED();
END_METHOD

END_FUNCTION_BLOCK

// ---- Tests/StackForwardEnumerator_TestSuite.TcPOU
FUNCTION_BLOCK PUBLIC StackForwardEnumerator_TestSuite EXTENDS TcUnit.FB_TestSuite

CheckIsValidAtStart();
CheckMoveNextReturnsFalseAtTheEnd();
CheckMoveNextReturnsFalseWhenEmpty();
CheckMoveNextReturnsTrueMultipleItems();
CheckMoveNextReturnsTrueSingleItem();
CheckReset();
CheckTryGet();
CheckTryGetTo();
CheckWorksWithIntegers();
CheckWorksWithStrings();
CheckWorksWithArrays();

METHOD PUBLIC CheckIsValidAtStart
VAR
	result : BOOL;
	stack : Stack;
	enumerator : I_ForwardEnumerator;
END_VAR
TEST('CheckIsValidAtStart');

enumerator := stack.GetEnumerator();

result := enumerator.IsValid;
enumerator.Dispose();

AssertTrue(
	Condition := result,
	Message := 'Method returned false'
);

TEST_FINISHED();
END_METHOD

METHOD PRIVATE CheckMoveNextReturnsFalseAtTheEnd
VAR
	in1 : INT := 123;
	result : BOOL;
	stack : Stack;
	enumerator : I_ForwardEnumerator;
END_VAR
TEST('CheckMoveNextReturnsFalseAtTheEnd');

stack.Push(in1);
enumerator := stack.GetEnumerator();

enumerator.MoveNext();
result := enumerator.MoveNext();
enumerator.Dispose();

AssertFalse(result,
    'MoveNext did not correctly signal the end of the enumeration');
	
TEST_FINISHED();
END_METHOD

METHOD PUBLIC CheckMoveNextReturnsFalseWhenEmpty
VAR
	result : BOOL;
	stack : Stack;
	enumerator : I_ForwardEnumerator;
END_VAR
TEST('CheckMoveNextReturnsFalseWhenEmpty');

enumerator := stack.GetEnumerator();

result := enumerator.MoveNext();
enumerator.Dispose();

AssertFalse(
	Condition := result,
	Message := 'MoveNext did not correctly signal the end of the enumeration'
);

TEST_FINISHED();
END_METHOD

METHOD PRIVATE CheckMoveNextReturnsTrueMultipleItems
VAR
	in1 : INT := 123;
	in2 : INT := 456;
	in3 : INT := 789;
	result : BOOL;
	stack : Stack;
	enumerator : I_ForwardEnumerator;
END_VAR
TEST('CheckMoveNextReturnsTrueMultipleItems');

stack.Push(in1);
stack.Push(in2);
stack.Push(in3);
enumerator := stack.GetEnumerator();

result := enumerator.MoveNext();
enumerator.Dispose();

AssertTrue(result, 'MoveNext did not correctly signal there were more items to follow');

TEST_FINISHED();
END_METHOD

METHOD PRIVATE CheckMoveNextReturnsTrueSingleItem
VAR
	in1 : INT := 123;
	result : BOOL;
	stack : Stack;
	enumerator : I_ForwardEnumerator;
END_VAR
TEST('CheckMoveNextReturnsTrueSingleItem');

stack.Push(in1);
enumerator := stack.GetEnumerator();

result := enumerator.MoveNext();
enumerator.Dispose();

AssertTrue(result,
    'MoveNext did not correctly signal there were more items to follow');
	
TEST_FINISHED();
END_METHOD

METHOD PUBLIC CheckReset
VAR
	in1 : ARRAY [0..1] OF REAL := [0.1,2.3];
	in2 : ARRAY [0..1] OF REAL := [1.2,3.4];
	in3 : ARRAY [0..1] OF REAL := [2.3,4.5];
	out : ARRAY [0..1] OF REAL;
	expected : ARRAY [0..1] OF REAL := [2.3,4.5];
	stack : Stack;
	enumerator : I_ForwardEnumerator;
END_VAR
TEST('CheckReset');

stack.Push(in1);
stack.Push(in2);
stack.Push(in3);

enumerator := stack.GetEnumerator();

enumerator.MoveNext();
enumerator.MoveNext();
enumerator.Reset();
enumerator.MoveNext();
enumerator.TryGet(out);

enumerator.Dispose();

AssertEquals(
	Expected := expected,
	Actual := out,
	Message := 'Did not produce the expected result'
);

TEST_FINISHED();
END_METHOD

METHOD PUBLIC CheckTryGet
VAR
	in : INT := 123;
	out : INT;
	expected : INT := 123;
	result : BOOL;
	stack : Stack;
	enumerator : I_ForwardEnumerator;
END_VAR
TEST('CheckTryGet');

stack.Push(in);
enumerator := stack.GetEnumerator();
enumerator.MoveNext();

result := enumerator.TryGet(out);
enumerator.Dispose();

AssertTrue(
	Condition := result,
	Message := 'Method returned false'
);

AssertEquals(
	Expected := expected,
	Actual := out,
	Message := 'Did not produce the expected result'
);

TEST_FINISHED();
END_METHOD

METHOD PUBLIC CheckTryGetTo
VAR
	in : INT := 123;
	out : INT;
	expected : INT := 123;
	result : BOOL;
	stack : Stack;
	enumerator : I_ForwardEnumerator;
END_VAR
TEST('CheckTryGetTo');

stack.Push(in);
enumerator := stack.GetEnumerator();
enumerator.MoveNext();

result := enumerator.TryGetTo(ADR(out),SIZEOF(out));
enumerator.Dispose();

AssertTrue(
	Condition := result,
	Message := 'Method returned false'
);

AssertEquals(
	Expected := expected,
	Actual := out,
	Message := 'Did not produce the expected result'
);

TEST_FINISHED();
END_METHOD

METHOD PUBLIC CheckWorksWithArrays
VAR
	in1 : ARRAY [0..1] OF REAL := [0.1,2.3];
	in2 : ARRAY [0..1] OF REAL := [1.2,3.4];
	in3 : ARRAY [0..1] OF REAL := [2.3,4.5];
	out1 : ARRAY [0..1] OF REAL;
	out2 : ARRAY [0..1] OF REAL;
	out3 : ARRAY [0..1] OF REAL;
	expected1 : ARRAY [0..1] OF REAL := [2.3,4.5];
	expected2 : ARRAY [0..1] OF REAL := [1.2,3.4];
	expected3 : ARRAY [0..1] OF REAL := [0.1,2.3];
	stack : Stack;
	enumerator : I_ForwardEnumerator;
END_VAR
TEST('CheckWorksWithArrays');

stack.Push(in1);
stack.Push(in2);
stack.Push(in3);

enumerator := stack.GetEnumerator();

enumerator.MoveNext();
enumerator.TryGet(out1);
enumerator.MoveNext();
enumerator.TryGet(out2);
enumerator.MoveNext();
enumerator.TryGet(out3);

enumerator.Dispose();

AssertEquals(
	Expected := expected1,
	Actual := out1,
	Message := 'Did not produce the expected 1st result'
);

AssertEquals(
	Expected := expected2,
	Actual := out2,
	Message := 'Did not produce the expected 2nd result'
);

AssertEquals(
	Expected := expected3,
	Actual := out3,
	Message := 'Did not produce the expected 3rd result'
);

TEST_FINISHED();
END_METHOD

METHOD PUBLIC CheckWorksWithIntegers
VAR
	in1 : INT := 123;
	in2 : INT := 234;
	in3 : INT := 345;
	out1 : INT;
	out2 : INT;
	out3 : INT;
	expected1 : INT := 345;
	expected2 : INT := 234;
	expected3 : INT := 123;
	stack : Stack;
	enumerator : I_ForwardEnumerator;
END_VAR
TEST('CheckWorksWithIntegers');

stack.Push(in1);
stack.Push(in2);
stack.Push(in3);

enumerator := stack.GetEnumerator();

enumerator.MoveNext();
enumerator.TryGet(out1);
enumerator.MoveNext();
enumerator.TryGet(out2);
enumerator.MoveNext();
enumerator.TryGet(out3);

enumerator.Dispose();

AssertEquals(
	Expected := expected1,
	Actual := out1,
	Message := 'Did not produce the expected 1st result'
);

AssertEquals(
	Expected := expected2,
	Actual := out2,
	Message := 'Did not produce the expected 2nd result'
);

AssertEquals(
	Expected := expected3,
	Actual := out3,
	Message := 'Did not produce the expected 3rd result'
);

TEST_FINISHED();
END_METHOD

METHOD PUBLIC CheckWorksWithStrings
VAR
	in1 : STRING := 'test1';
	in2 : STRING := 'test2';
	in3 : STRING := 'test3';
	out1 : STRING;
	out2 : STRING;
	out3 : STRING;
	expected1 : STRING := 'test3';
	expected2 : STRING := 'test2';
	expected3 : STRING := 'test1';
	stack : Stack;
	enumerator : I_ForwardEnumerator;
END_VAR
TEST('CheckWorksWithStrings');

stack.Push(in1);
stack.Push(in2);
stack.Push(in3);

enumerator := stack.GetEnumerator();

enumerator.MoveNext();
enumerator.TryGet(out1);
enumerator.MoveNext();
enumerator.TryGet(out2);
enumerator.MoveNext();
enumerator.TryGet(out3);

enumerator.Dispose();

AssertEquals(
	Expected := expected1,
	Actual := out1,
	Message := 'Did not produce the expected 1st result'
);

AssertEquals(
	Expected := expected2,
	Actual := out2,
	Message := 'Did not produce the expected 2nd result'
);

AssertEquals(
	Expected := expected3,
	Actual := out3,
	Message := 'Did not produce the expected 3rd result'
);

TEST_FINISHED();
END_METHOD

END_FUNCTION_BLOCK
